FUNCTION_BLOCK TCounter
VAR
    Count : DINT;
END_VAR

METHOD Dec : DINT
VAR_INPUT
END_VAR
Count := Count - 1;
Dec := Count;
END_METHOD

METHOD Inc : DINT
VAR_INPUT
END_VAR
Count := Count + 1;
Inc := Count;
END_METHOD

METHOD Reset
VAR_INPUT
END_VAR
Count := 0;
END_METHOD

PROPERTY Value : DINT
GET
Value := Count;
END_GET
SET
Count := Value;
END_SET
END_PROPERTY

PROPERTY ValueAsTArg : T_Arg
GET
ValueAsTArg := F_DINT(Count);
END_GET
END_PROPERTY

END_FUNCTION_BLOCK

(* stored: Version 1.1.0.1, ProductVersion 3.1.4024.3
   POU TCounter: Id {efd6445c-34ee-479f-8c19-794d742925a3}, SpecialFunc None
   Method Dec: Id {c442b024-7db9-41cf-99c4-34cf96c9c66d}
   Method Inc: Id {2ca2f8ff-5d58-4fe6-837c-d61767ce93e0}
   Method Reset: Id {befc5dfc-e327-4e0c-a1ca-6ff557cccbf4}
   Property Value: Id {9c6285da-44cf-4672-892f-bd3c9a26ffa1}
   Get Get: Id {c79fc04b-5b1a-4fd1-8a40-bf12c9ea808b}
   Set Set: Id {b4985470-e595-436b-b429-7a7739ae4d85}
   Property ValueAsTArg: Id {c11a11e6-00a7-44f7-bb4b-a531326ce700}
   Get Get: Id {dcfdbc27-88ef-45a3-b319-0c7b531fd7d8} *)
